{attribute addProperty BoxType "EP6224-2022-0018"}
{attribute addProperty Id "Module_1_DeviceState_Inputs_DeviceModule_1_DeviceState_Inputs_Device_50DD3C951620Module_2_DeviceState_InputsModule_2_DeviceState_Inputs_D860B2E33240WcStateAT %I*WcState_98A4DF7520.250InfoDataAT %I*InfoData_275E3363128160"}
{attribute addProperty CRC "1978599132"}
{attribute addProperty SizeInBites "178"}
{attribute addProperty SizeInBytes "22.25"}
TYPE EP6224_3990B4B4 :
STRUCT
	{attribute addProperty Name "Module_1_DeviceState_Inputs_Device"}
	Module_1_DeviceState_Inputs_Device : Module_1_DeviceState_Inputs_Device_50DD3C95;
	{attribute addProperty Name "Module_2_DeviceState_Inputs"}
	Module_2_DeviceState_Inputs : Module_2_DeviceState_Inputs_D860B2E3;
	{attribute addProperty Name "WcState"}
	WcState : WcState_98A4DF75;
	{attribute addProperty Name "InfoData"}
	InfoData : InfoData_275E3363;
END_STRUCT
END_TYPE

(* stored: Version 1.2.0.0, ProductVersion 3.1.4024.9
   DUT EP6224_3990B4B4: Id {d5e5456b-e0c9-4fb4-b65f-73a5bbc8be8a} *)
